{attribute 'TcGenerated'}
// This function has been automatically generated from the project information.
VAR_GLOBAL CONSTANT
    {attribute 'const_non_replaced'}
    {attribute 'linkalways'}
    stLibVersion_lcls_plc_lfe_optics : ST_LibVersion := (iMajor := 1, iMinor := 2, iBuild := 0, iRevision := 0, sVersion := '1.2.0');
END_VAR

(* stored: Version 1.1.0.1, ProductVersion 3.1.4022.18
   GVL Global_Version: Id 679697c4-2481-46d4-a3fd-e071ccb7400e *)
